// TIA Portal project "assemble" (V17)
// Vorlageprojekt für das Buch mit Zielsystem S7-1200

(* hardware
DEVICE "S7-1200-Station_1"  S7-1200 Station
   slot 0: "Baugruppenträger_0"  Rack  V1.0
   slot 1: "PLC_1"  CPU 1211C DC/DC/DC  6ES7 211-1AE40-0XB0  V4.1
*)

// ===== PLC "PLC_1"  CPU 1211C DC/DC/DC =====

VAR_GLOBAL   // PLC tag table "Standard-Variablentabelle"
   "lid at place" AT %I0.3 : Bool;
   "move x" AT %E0.0 : Bool;
   "move y" AT %E0.1 : Bool;
   "item detected" AT %I0.2 : Bool;
   "clamp at max (lid)" AT %I0.5 : Bool;
   "base at place" AT %I0.6 : Bool;
   "lid clamed" AT %I0.4 : Bool;
   "base clamed" AT %I0.7 : Bool;
   "clamp at max (base)" AT %I1.0 : Bool;
   "counter" AT %QD30 : DWord;
   "part leaveing" AT %I1.1 : Bool;
   "start" AT %I1.2 : Bool;
   "reset" AT %I1.3 : Bool;
   "stop" AT %I1.4 : Bool;
   "emergency stop" AT %I1.5 : Bool;
   "auto" AT %I1.6 : Bool;
   "move x(1)" AT %Q0.0 : Bool;
   "move y(1)" AT %Q0.1 : Bool;
   "grab" AT %Q0.2 : Bool;
   "conveyor lid" AT %Q0.3 : Bool;
   "clamp lid" AT %Q0.4 : Bool;
   "clamp raised (lid)" AT %Q0.5 : Bool;
   "conveyor base" AT %Q0.6 : Bool;
   "clamp base" AT %Q0.7 : Bool;
   "clamp raised (base)" AT %Q1.0 : Bool;
   "start light" AT %Q1.1 : Bool;
   "reset light" AT %Q1.2 : Bool;
   "stop light" AT %Q1.3 : Bool;
   "Tag_1" AT %M0.3 : Bool;
   "Tag_2" AT %M0.6 : Bool;
   "Tag_3" AT %M1.1 : Bool;
   "Tag_4" AT %M0.4 : Bool;
   "lid alinde" AT %M1.7 : Bool;
   "Tag_5" AT %M1.0 : Bool;
   "Tag_6" AT %M0.7 : Bool;
   "base alinde" AT %M1.6 : Bool;
   "Tag_7" AT %M0.0 : Bool;
   "Tag_8" AT %M0.1 : Bool;
   "Tag_9" AT %M0.2 : Bool;
   "move lid" AT %M1.5 : Bool;
   "Tag_10" AT %M0.5 : Bool;
   "Tag_11" AT %M1.4 : Bool;
   "Tag_12" AT %M1.3 : Bool;
   "Tag_13" AT %M1.2 : Bool;
   "Tag_14" AT %M2.0 : Bool;
   "move lid2" AT %M2.1 : Bool;
   "Tag_15" AT %M2.2 : Bool;
   "temporar" AT %M2.3 : Bool;
   "Tag_16" AT %M2.4 : Bool;
   "temp2" AT %M2.5 : Bool;
   "Tag_17" AT %M2.6 : Bool;
END_VAR

// folder: System blocks/Program resources

DATA_BLOCK "IEC_Timer_0_DB"   // DB1
{ S7_Optimized_Access := 'TRUE' }
AUTHOR : Simatic
FAMILY : IEC
NAME : IEC_TMR
VERSION : 1.0
// stored: InstanceOfName IEC_TIMER
"IEC_TIMER"
BEGIN
END_DATA_BLOCK

DATA_BLOCK "IEC_Timer_0_DB_1"   // DB2
{ S7_Optimized_Access := 'TRUE' }
AUTHOR : Simatic
FAMILY : IEC
NAME : IEC_TMR
VERSION : 1.0
// stored: InstanceOfName IEC_TIMER
"IEC_TIMER"
BEGIN
END_DATA_BLOCK

DATA_BLOCK "IEC_Timer_0_DB_2"   // DB3
{ S7_Optimized_Access := 'TRUE' }
AUTHOR : Simatic
FAMILY : IEC
NAME : IEC_TMR
VERSION : 1.0
// stored: InstanceOfName IEC_TIMER
"IEC_TIMER"
BEGIN
END_DATA_BLOCK

// folder: (top level)

FUNCTION "conveyor" : Void   // FC1, LAD
{ S7_Optimized_Access := 'TRUE' }
VERSION : 0.1
   VAR_TEMP   // added for the SCL form of the ladder/FBD networks
      _w1 : Bool;
   END_VAR
BEGIN

REGION Network 1
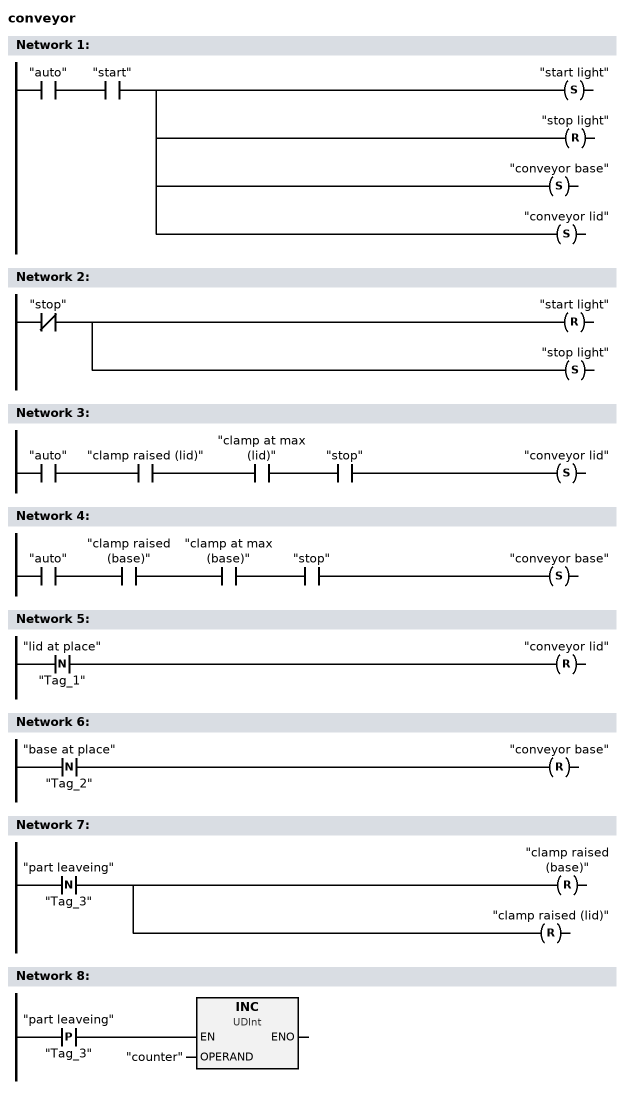
   RUNG wire#powerrail
      Contact( "auto" )
      Contact( "start" )
      wire#w1
      S_Coil( "start light" )
   END_RUNG
   RUNG wire#w1
      R_Coil( "stop light" )
   END_RUNG
   RUNG wire#w1
      S_Coil( "conveyor base" )
   END_RUNG
   RUNG wire#w1
      S_Coil( "conveyor lid" )
   END_RUNG
   // the same network as SCL:
   IF "auto" AND "start" THEN
       "start light" := TRUE;
       "stop light" := FALSE;
       "conveyor base" := TRUE;
       "conveyor lid" := TRUE;
   END_IF;
END_REGION

REGION Network 2
   RUNG wire#powerrail
      I_Contact( "stop" )
      wire#w1
      R_Coil( "start light" )
   END_RUNG
   RUNG wire#w1
      S_Coil( "stop light" )
   END_RUNG
   // the same network as SCL:
   IF NOT "stop" THEN
       "start light" := FALSE;
       "stop light" := TRUE;
   END_IF;
END_REGION

REGION Network 3
   RUNG wire#powerrail
      Contact( "auto" )
      Contact( "clamp raised (lid)" )
      Contact( "clamp at max (lid)" )
      Contact( "stop" )
      S_Coil( "conveyor lid" )
   END_RUNG
   // the same network as SCL:
   IF "auto" AND "clamp raised (lid)" AND "clamp at max (lid)" AND "stop" THEN
       "conveyor lid" := TRUE;
   END_IF;
END_REGION

REGION Network 4
   RUNG wire#powerrail
      Contact( "auto" )
      Contact( "clamp raised (base)" )
      Contact( "clamp at max (base)" )
      Contact( "stop" )
      S_Coil( "conveyor base" )
   END_RUNG
   // the same network as SCL:
   IF "auto" AND "clamp raised (base)" AND "clamp at max (base)" AND "stop" THEN
       "conveyor base" := TRUE;
   END_IF;
END_REGION

REGION Network 5
   RUNG wire#powerrail
      N_Contact(operand := "lid at place", bit := "Tag_1")
      R_Coil( "conveyor lid" )
   END_RUNG
   // the same network as SCL:
   #_w1 := NOT "lid at place" AND "Tag_1";   // falling edge of "lid at place"
   "Tag_1" := "lid at place";
   IF #_w1 THEN "conveyor lid" := FALSE; END_IF;
END_REGION

REGION Network 6
   RUNG wire#powerrail
      N_Contact(operand := "base at place", bit := "Tag_2")
      R_Coil( "conveyor base" )
   END_RUNG
   // the same network as SCL:
   #_w1 := NOT "base at place" AND "Tag_2";   // falling edge of "base at place"
   "Tag_2" := "base at place";
   IF #_w1 THEN "conveyor base" := FALSE; END_IF;
END_REGION

REGION Network 7
   RUNG wire#powerrail
      N_Contact(operand := "part leaveing", bit := "Tag_3")
      wire#w1
      R_Coil( "clamp raised (base)" )
   END_RUNG
   RUNG wire#w1
      R_Coil( "clamp raised (lid)" )
   END_RUNG
   // the same network as SCL:
   #_w1 := NOT "part leaveing" AND "Tag_3";   // falling edge of "part leaveing"
   "Tag_3" := "part leaveing";
   IF #_w1 THEN
       "clamp raised (base)" := FALSE;
       "clamp raised (lid)" := FALSE;
   END_IF;
END_REGION

REGION Network 8
   RUNG wire#powerrail
      P_Contact(operand := "part leaveing", bit := "Tag_3")
      { S7_Templates := "DestType := UDInt" } Inc( "counter" )
   END_RUNG
   // the same network as SCL:
   #_w1 := "part leaveing" AND NOT "Tag_3";   // rising edge of "part leaveing"
   "Tag_3" := "part leaveing";
   IF #_w1 THEN "counter" := "counter" + 1; END_IF;
END_REGION
END_FUNCTION

FUNCTION "clamp" : Void   // FC2, LAD
{ S7_Optimized_Access := 'TRUE' }
VERSION : 0.1
   VAR_TEMP   // added for the SCL form of the ladder/FBD networks
      _w1 : Bool;
   END_VAR
BEGIN

REGION Network 1
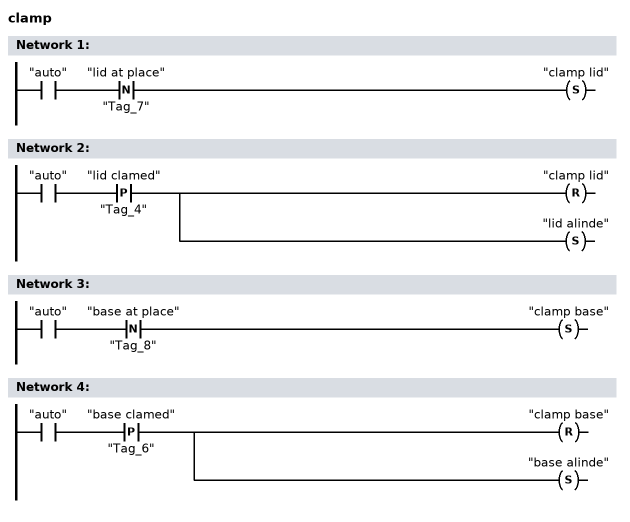
   RUNG wire#powerrail
      Contact( "auto" )
      N_Contact(operand := "lid at place", bit := "Tag_7")
      S_Coil( "clamp lid" )
   END_RUNG
   // the same network as SCL:
   #_w1 := "auto" AND NOT "lid at place" AND "Tag_7";   // falling edge of "lid at place"
   "Tag_7" := "lid at place";
   IF #_w1 THEN "clamp lid" := TRUE; END_IF;
END_REGION

REGION Network 2
   RUNG wire#powerrail
      Contact( "auto" )
      P_Contact(operand := "lid clamed", bit := "Tag_4")
      wire#w1
      R_Coil( "clamp lid" )
   END_RUNG
   RUNG wire#w1
      S_Coil( "lid alinde" )
   END_RUNG
   // the same network as SCL:
   #_w1 := "auto" AND "lid clamed" AND NOT "Tag_4";   // rising edge of "lid clamed"
   "Tag_4" := "lid clamed";
   IF #_w1 THEN
       "clamp lid" := FALSE;
       "lid alinde" := TRUE;
   END_IF;
END_REGION

REGION Network 3
   RUNG wire#powerrail
      Contact( "auto" )
      N_Contact(operand := "base at place", bit := "Tag_8")
      S_Coil( "clamp base" )
   END_RUNG
   // the same network as SCL:
   #_w1 := "auto" AND NOT "base at place" AND "Tag_8";   // falling edge of "base at place"
   "Tag_8" := "base at place";
   IF #_w1 THEN "clamp base" := TRUE; END_IF;
END_REGION

REGION Network 4
   RUNG wire#powerrail
      Contact( "auto" )
      P_Contact(operand := "base clamed", bit := "Tag_6")
      wire#w1
      R_Coil( "clamp base" )
   END_RUNG
   RUNG wire#w1
      S_Coil( "base alinde" )
   END_RUNG
   // the same network as SCL:
   #_w1 := "auto" AND "base clamed" AND NOT "Tag_6";   // rising edge of "base clamed"
   "Tag_6" := "base clamed";
   IF #_w1 THEN
       "clamp base" := FALSE;
       "base alinde" := TRUE;
   END_IF;
END_REGION
END_FUNCTION

FUNCTION "pick_and_move" : Void   // FC3, LAD
{ S7_Optimized_Access := 'TRUE' }
VERSION : 0.1
   VAR_TEMP   // added for the SCL form of the ladder/FBD networks
      _w1 : Bool;
   END_VAR
BEGIN

REGION Network 1
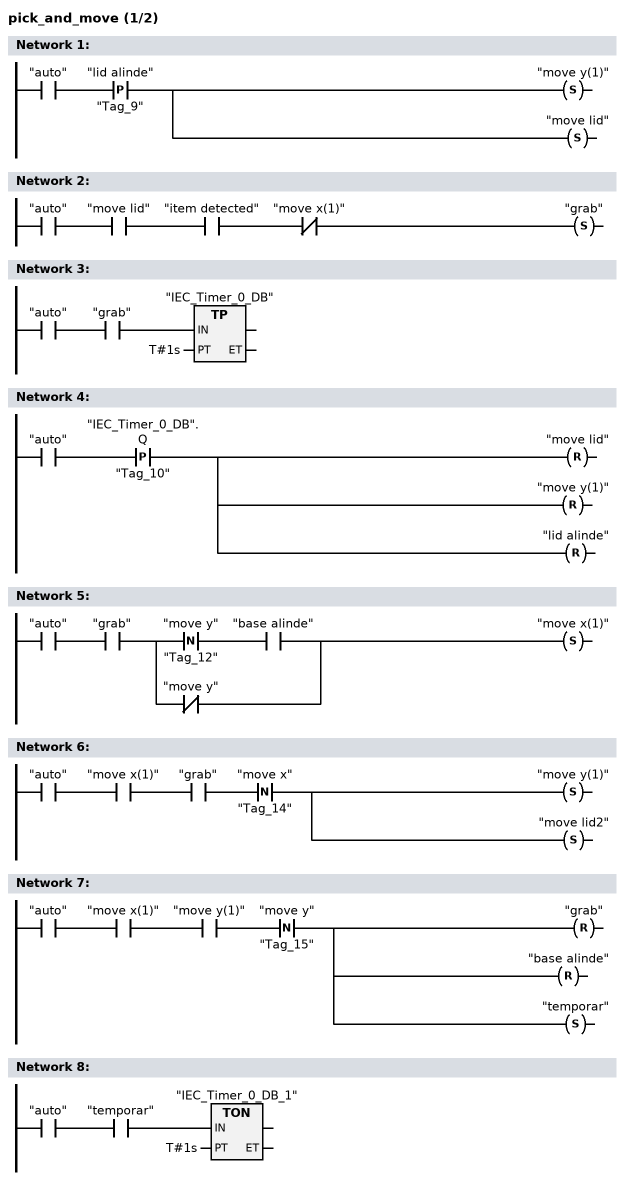
   RUNG wire#powerrail
      Contact( "auto" )
      P_Contact(operand := "lid alinde", bit := "Tag_9")
      wire#w1
      S_Coil( "move y(1)" )
   END_RUNG
   RUNG wire#w1
      S_Coil( "move lid" )
   END_RUNG
   // the same network as SCL:
   #_w1 := "auto" AND "lid alinde" AND NOT "Tag_9";   // rising edge of "lid alinde"
   "Tag_9" := "lid alinde";
   IF #_w1 THEN
       "move y(1)" := TRUE;
       "move lid" := TRUE;
   END_IF;
END_REGION

REGION Network 2
   RUNG wire#powerrail
      Contact( "auto" )
      Contact( "move lid" )
      Contact( "item detected" )
      I_Contact( "move x(1)" )
      S_Coil( "grab" )
   END_RUNG
   // the same network as SCL:
   IF "auto" AND "move lid" AND "item detected" AND NOT "move x(1)" THEN "grab" := TRUE; END_IF;
END_REGION

REGION Network 3
   "IEC_Timer_0_DB".TP(IN := "auto" AND "grab", PT := T#1s);
END_REGION

REGION Network 4
   RUNG wire#powerrail
      Contact( "auto" )
      P_Contact(operand := "IEC_Timer_0_DB".Q, bit := "Tag_10")
      wire#w1
      R_Coil( "move lid" )
   END_RUNG
   RUNG wire#w1
      R_Coil( "move y(1)" )
   END_RUNG
   RUNG wire#w1
      R_Coil( "lid alinde" )
   END_RUNG
   // the same network as SCL:
   #_w1 := "auto" AND "IEC_Timer_0_DB".Q AND NOT "Tag_10";   // rising edge of "IEC_Timer_0_DB".Q
   "Tag_10" := "IEC_Timer_0_DB".Q;
   IF #_w1 THEN
       "move lid" := FALSE;
       "move y(1)" := FALSE;
       "lid alinde" := FALSE;
   END_IF;
END_REGION

REGION Network 5
   RUNG wire#powerrail
      Contact( "auto" )
      Contact( "grab" )
      wire#w1
      N_Contact(operand := "move y", bit := "Tag_12")
      Contact( "base alinde" )
      wire#w2
      S_Coil( "move x(1)" )
   END_RUNG
   RUNG wire#w1
      I_Contact( "move y" )
   END_RUNG wire#w2
   // the same network as SCL:
   #_w1 := "auto" AND "grab" AND NOT "move y" AND "Tag_12";   // falling edge of "move y"
   "Tag_12" := "move y";
   IF (#_w1 AND "base alinde") OR ("auto" AND "grab" AND NOT "move y") THEN "move x(1)" := TRUE; END_IF;
END_REGION

REGION Network 6
   RUNG wire#powerrail
      Contact( "auto" )
      Contact( "move x(1)" )
      Contact( "grab" )
      N_Contact(operand := "move x", bit := "Tag_14")
      wire#w1
      S_Coil( "move y(1)" )
   END_RUNG
   RUNG wire#w1
      S_Coil( "move lid2" )
   END_RUNG
   // the same network as SCL:
   #_w1 := "auto" AND "move x(1)" AND "grab" AND NOT "move x" AND "Tag_14";   // falling edge of "move x"
   "Tag_14" := "move x";
   IF #_w1 THEN
       "move y(1)" := TRUE;
       "move lid2" := TRUE;
   END_IF;
END_REGION

REGION Network 7
   RUNG wire#powerrail
      Contact( "auto" )
      Contact( "move x(1)" )
      Contact( "move y(1)" )
      N_Contact(operand := "move y", bit := "Tag_15")
      wire#w1
      R_Coil( "grab" )
   END_RUNG
   RUNG wire#w1
      R_Coil( "base alinde" )
   END_RUNG
   RUNG wire#w1
      S_Coil( "temporar" )
   END_RUNG
   // the same network as SCL:
   #_w1 := "auto" AND "move x(1)" AND "move y(1)" AND NOT "move y" AND "Tag_15";   // falling edge of "move y"
   "Tag_15" := "move y";
   IF #_w1 THEN
       "grab" := FALSE;
       "base alinde" := FALSE;
       "temporar" := TRUE;
   END_IF;
END_REGION

REGION Network 8
   "IEC_Timer_0_DB_1".TON(IN := "auto" AND "temporar", PT := T#1s);
END_REGION

REGION Network 9
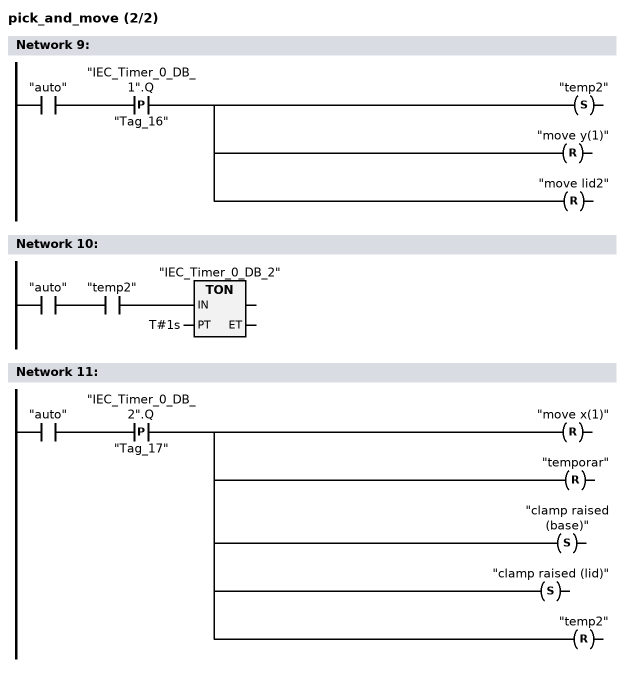
   RUNG wire#powerrail
      Contact( "auto" )
      P_Contact(operand := "IEC_Timer_0_DB_1".Q, bit := "Tag_16")
      wire#w1
      S_Coil( "temp2" )
   END_RUNG
   RUNG wire#w1
      R_Coil( "move y(1)" )
   END_RUNG
   RUNG wire#w1
      R_Coil( "move lid2" )
   END_RUNG
   // the same network as SCL:
   #_w1 := "auto" AND "IEC_Timer_0_DB_1".Q AND NOT "Tag_16";   // rising edge of "IEC_Timer_0_DB_1".Q
   "Tag_16" := "IEC_Timer_0_DB_1".Q;
   IF #_w1 THEN
       "temp2" := TRUE;
       "move y(1)" := FALSE;
       "move lid2" := FALSE;
   END_IF;
END_REGION

REGION Network 10
   "IEC_Timer_0_DB_2".TON(IN := "auto" AND "temp2", PT := T#1s);
END_REGION

REGION Network 11
   RUNG wire#powerrail
      Contact( "auto" )
      P_Contact(operand := "IEC_Timer_0_DB_2".Q, bit := "Tag_17")
      wire#w1
      R_Coil( "move x(1)" )
   END_RUNG
   RUNG wire#w1
      R_Coil( "temporar" )
   END_RUNG
   RUNG wire#w1
      S_Coil( "clamp raised (base)" )
   END_RUNG
   RUNG wire#w1
      S_Coil( "clamp raised (lid)" )
   END_RUNG
   RUNG wire#w1
      R_Coil( "temp2" )
   END_RUNG
   // the same network as SCL:
   #_w1 := "auto" AND "IEC_Timer_0_DB_2".Q AND NOT "Tag_17";   // rising edge of "IEC_Timer_0_DB_2".Q
   "Tag_17" := "IEC_Timer_0_DB_2".Q;
   IF #_w1 THEN
       "move x(1)" := FALSE;
       "temporar" := FALSE;
       "clamp raised (base)" := TRUE;
       "clamp raised (lid)" := TRUE;
       "temp2" := FALSE;
   END_IF;
END_REGION
END_FUNCTION

FUNCTION "MHJ-PLC-Lab-Function-S71200" : Void   // FC9000, SCL
{ S7_Optimized_Access := 'TRUE' }
VERSION : 0.1
   VAR_TEMP
      rdTimeReturn : Int;
      outputTime : DTL;
      SyncVal : Byte;
      forVal : Int;
      forVal_2 : Int;
      Value : Byte;
   END_VAR
   VAR CONSTANT
      CompVal : Byte := 16#34;
      Value_01 : Byte := 16#11;
      Value_01_DW : DWord := 16#A165_D992;
      Value_02_DW : DWord := 16#58BE_4401;
   END_VAR
BEGIN

   #Value:=PEEK(area := 16#82,
        dbNumber := 0,
        byteOffset := 511);
   #Value := #Value + 1;

   POKE(area := 16#82,
        dbNumber := 0,
        byteOffset := 511,
        value := #Value);

   POKE(area:=16#81,
        dbNumber:=0,
        byteOffset:=1016,
        value:=#Value_01_DW);
   POKE(area := 16#81,
        dbNumber := 0,
        byteOffset := 1020,
        value := #Value_02_DW);

   POKE(area := 16#81,
        dbNumber := 0,
        byteOffset := 511,
        value := B#16#00);

   FOR #forVal := 0 TO 120 DO
       FOR #forVal_2:=0 TO 10 DO
           #rdTimeReturn:=RD_SYS_T(#outputTime);
           #rdTimeReturn := WR_SYS_T(#outputTime);
           #rdTimeReturn := RD_SYS_T(#outputTime);
           #rdTimeReturn := WR_SYS_T(#outputTime);
       END_FOR;
       #SyncVal:= PEEK(area := 16#81,
                      dbNumber := 0,
                      byteOffset := 511);
       IF #SyncVal = #CompVal THEN
          GOTO M_1;
       END_IF;
   END_FOR;
   RETURN;

   M_1:
   POKE(area := 16#81,
        dbNumber := 0,
        byteOffset := 511,
        value := B#16#0);
END_FUNCTION

ORGANIZATION_BLOCK "Main"   // OB1, FBD, ProgramCycle
TITLE = "Main Program Sweep (Cycle)"
{ S7_Optimized_Access := 'TRUE' }
VERSION : 0.1
   VAR_INPUT
      Initial_Call : Bool;   // Initial call of this OB
      Remanence : Bool;   // =True, if remanent data are available
   END_VAR
BEGIN

REGION Network 1: Konnektierungsbaustein für PLC-Lab
   // Im Netzwerk 1 wird der Konnektierungsbaustein für PLC-Lab aufgerufen.
   // Dieser Aufruf darf nicht entfernt werden!
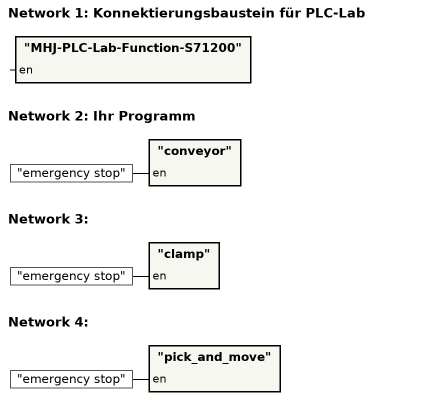
   "MHJ-PLC-Lab-Function-S71200"();
END_REGION

REGION Network 2: Ihr Programm
   // Schreiben Sie ab Netzwerk 2 Ihr Programm
   IF "emergency stop" THEN "conveyor"(); END_IF;
END_REGION

REGION Network 3
   IF "emergency stop" THEN "clamp"(); END_IF;
END_REGION

REGION Network 4
   IF "emergency stop" THEN "pick_and_move"(); END_IF;
END_REGION
END_ORGANIZATION_BLOCK